{attribute 'GeneratedUsingTerminal: ELM3002-0000-0016'}
{attribute addProperty BoxType "ELM3002-0000-0016"}
{attribute addProperty Id "SamplesAT %I*Samples_F24E104A4"}
{attribute addProperty CRC "4003796773"}
{attribute addProperty Size "4"}
TYPE PAI_Samples_1_Channel_EEA51725 :
STRUCT
	{attribute addProperty Name "Samples"}
	Samples AT %I* : Samples_F24E104A;
END_STRUCT
END_TYPE

(* stored: Version 1.2.0.0, ProductVersion 3.1.4024.9
   DUT PAI_Samples_1_Channel_EEA51725: Id {8de419be-80c5-4625-b6b8-00291cd4607f} *)
